// TIA Portal V16 export
// export: Created 2023-08-28T09:37:54.601879Z, ExportSetting WithDefaults, DisplayName Totally Integrated Automation Portal, DisplayVersion V16 Update 6, DisplayName TIA Portal Version Control Interface, DisplayVersion V16 Update 2, DisplayName TIA Portal Openness, DisplayVersion V16 Update 6, DisplayName STEP 7 Professional, DisplayVersion V16 Update 6, DisplayName STEP 7 Safety, DisplayVersion V16, DisplayName WinCC Advanced, DisplayVersion V16 Update 6
VAR_GLOBAL   // PLC tag table "P4"
   inputRunF_P4 AT %M81.3 : Bool;   // stycznik falownik / Potwierdzenie pracy z falownika
   inputRunS_P4 AT %M80.7 : Bool;   // stycznik softstart / Powierdzenie pracy z sieci
   inputReadyP4 AT %M80.3 : Bool;   // sugnał gotowość / Gotowość napędu
   IsReady_P4 AT %M83.3 : Bool;   // Znacznik gotowości napędu
   IsRunInverter_P4 AT %M83.4 : Bool;   // Potwierdzenie pracy z falownika
   IsRunNetwork_P4 AT %M83.5 : Bool;   // Potwierdzenie pracy z sieci
   CMD_inverter_P4 AT %M83.6 : Bool;   // Stycznik Falownik
   CMD_network_P4 AT %M83.7 : Bool;   // Stycznik Sieć
   CMD_soft_P4 AT %M85.2 : Bool;   // sygnał z softstart potwierdzenie pracy / sygnał on/off soft-start
   setCMD_FP4 AT %M87.0 : Bool;   // Znacznik sterowania w trybie falownik dlaP1
   setCMD_SP4 AT %M87.1 : Bool;   // Znacznik sterowania w trybie sieć
   CB_CMD_P4 AT %M88.3 : Bool;   // Znacznik polecenia on/off przekaźnik napędu
   Set_HWork_P4 AT %M88.5 : Bool;   // Znacznik ustawienia aktywnej do pracy (po porównaniu liczników pracy)
   Is_extras_K1_P4 AT %M88.6 : Bool;   // Znacznik motor dodatkowy nr 1
   Set_50Hz_P4 AT %M89.0 : Bool;   // Znacznik pamięci podtrzymujący przełączenie na sieć
   setSUPV_FP4 AT %M89.3 : Bool;   // Znacznik polecenia startu z falownika
   IsRun_P4 AT %M89.4 : Bool;   // Potwierdzenie pracy
   setSUPV_SP4 AT %M89.5 : Bool;   // Znacznik polecenia startu z sieci
   Hour_Work_P4 AT %MD29 : DWord;   // Licznik pracy
   resetFault_SoftStart_P4 AT %M50.3 : Bool;   // sygnał resetu softstart
   bitH_Alarm_P4 AT %M66.0 : Bool;   // Alarm - kopia bitu z instancji statusu napędu
   bitH_rezerwa_P4 AT %M66.1 : Bool;   // rez
   bitH_REM_P4 AT %M66.2 : Bool;   // Zdalna - kopia bitu z instancji statusu napędu
   bitH_RUN_P4 AT %M66.3 : Bool;   // Praca - kopia bitu z instancji statusu napędu
   bitH_OFF_P4 AT %M66.4 : Bool;   // Polecenie OFF - kopia bitu z instancji statusu napędu
   bitH_ON_P4 AT %M66.5 : Bool;   // Polecenie ON - kopia bitu z instancji statusu napędu
   bitH_Res_P4 AT %M66.6 : Bool;   // Reset - kopia bitu z instancji statusu napędu
   bitH_Aut_Man_P4 AT %M66.7 : Bool;   // Aut=1 Man=0 - kopia bitu z instancji statusu napędu
   Is_extras_K3_P4 AT %M90.0 : Bool;   // Znacznik motor dodatkowy nr 3
   Is_extras_K2_P4 AT %M88.7 : Bool;   // Znacznik motor dodatkowy nr 2
   off_add_K1_P4 AT %M53.1 : Bool;   // sterowanie wyłączeniem selektywnym dodatkowej
   off_add_K2_P4 AT %M53.2 : Bool;   // sterowanie wyłączeniem selektywnym dodatkowej
   off_add_K3_P4 AT %M53.3 : Bool;   // sterowanie wyłączeniem selektywnym dodatkowej
   off_add_K4_P4 AT %M53.7 : Bool;   // sterowanie wyłączeniem selektywnym dodatkowej
   CMD_ErrorSet_NetworkP4 AT %M89.1 : Bool;   // Znacznik sterowania awaryjnego pracą pompy bez falownika
   Mem_Res_setCMD_MC_P4 AT %M89.2 : Bool;   // pamięć zbocza załączenia timera blokowania stycznika falowni P1
END_VAR
